INTERFACE I_Metadatum

METHOD PUBLIC Accept
VAR_INPUT
	Visitor : I_MetadataVisitor;
END_VAR
END_METHOD

METHOD PUBLIC AddDataAsMetadata : I_Metadata
VAR_INPUT
	Name : T_MAXSTRING;
	Data : I_Datatype;
END_VAR
END_METHOD

METHOD AddMetadata
VAR_INPUT
	Metadata : I_Metadata;
END_VAR
END_METHOD

PROPERTY PUBLIC HasMetadata : BOOL
GET
END_GET
END_PROPERTY

METHOD PUBLIC TryGetMetadataByName : BOOL
VAR_INPUT
	Name : T_MAXSTRING;
	Destination : REFERENCE TO I_Metadata;
END_VAR
END_METHOD

END_INTERFACE

(* stored: Version 1.1.0.1, ProductVersion 3.1.4024.12
   Itf I_Metadatum: Id {91f437e7-22ce-4a18-82a9-ffa0ed34169e}
   Method Accept: Id {14e9e0ea-2bc6-4c0c-aa73-789721725b7c}
   Method AddDataAsMetadata: Id {018d7e1b-7b59-4a7d-a768-40096184a489}
   Method AddMetadata: Id {1fd7cb94-de70-4016-8a78-91964b5a2603}
   Property HasMetadata: Id {51aec957-b54d-0cdb-3689-9f8339ce236a}
   Get Get: Id {a1396354-2d15-07e2-10f7-9b7f913e58f3}
   Method TryGetMetadataByName: Id {15454fbb-65cf-4875-8f88-8113171874e4} *)
